// TIA Portal V20 export
DATA_BLOCK "GLOBAL_IDENT_HMI_IF_DB"   // DB208
{ S7_Optimized_Access := 'TRUE' }
AUTHOR : Tesla
FAMILY : Ident
VERSION : 1.0
// stored: AutoNumber false, MemoryReserve 100
   VAR
      Reader { S7_SetPoint := 'True'} : Array[0.."No_Reader"] of "IDENT_RW_HMI_DAT_UDT";   // Data Erased On Tag Not Present / 数据 Erased 打开 Tag 没有 在
   END_VAR
BEGIN
END_DATA_BLOCK
